// SIMATIC S7-200 project (STEP 7-Micro/WIN), CPU 224 UN REL 02.01

ORGANIZATION_BLOCK 主程序:OB1
TITLE=程序注释
BEGIN
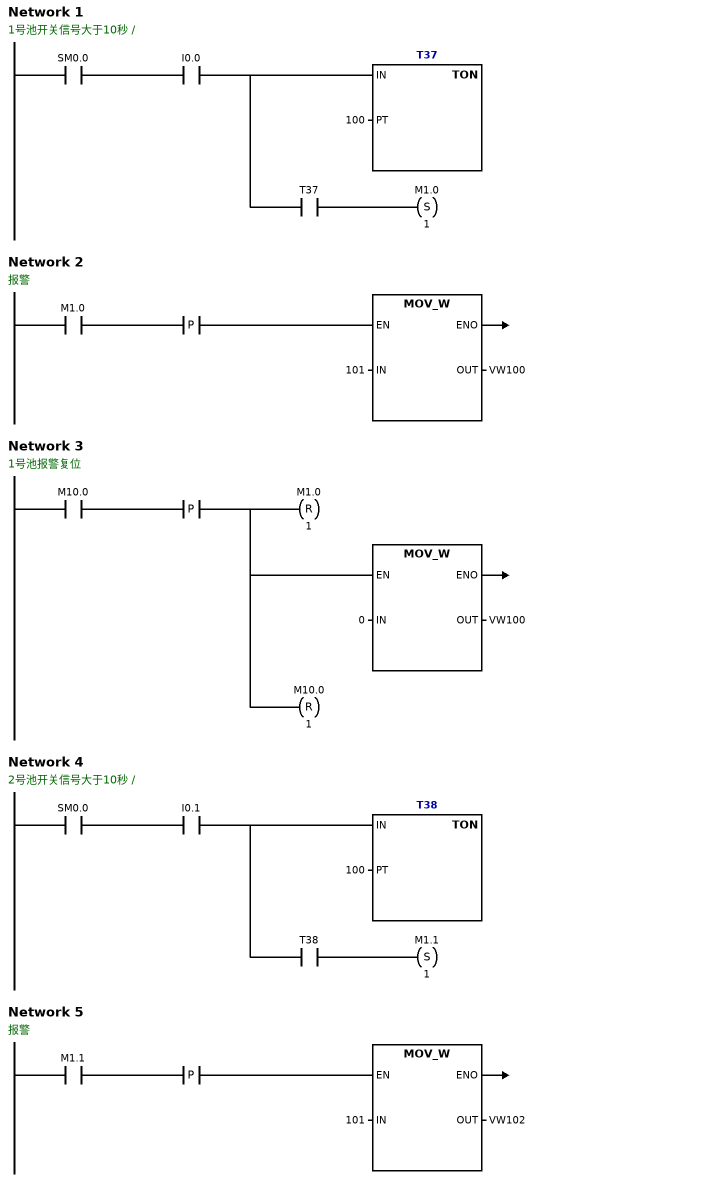
Network 1
// 1号池开关信号大于10秒
// 
LD     SM0.0
A      I0.0
TON    T37, 100
A      T37
S      M1.0, 1
Network 2 // 

// 报警
LD     M1.0
EU
MOVW   101, VW100
Network 3
// 1号池报警复位
LD     M10.0
EU
R      M1.0, 1
MOVW   0, VW100
R      M10.0, 1
Network 4
// 2号池开关信号大于10秒
// 
LD     SM0.0
A      I0.1
TON    T38, 100
A      T38
S      M1.1, 1
Network 5 // 

// 报警
LD     M1.1
EU
MOVW   101, VW102
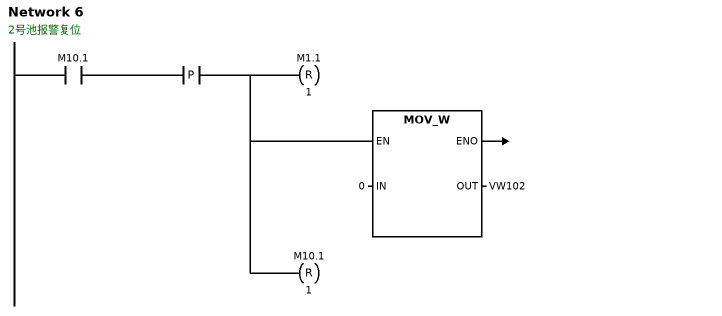
Network 6
// 2号池报警复位
LD     M10.1
EU
R      M1.1, 1
MOVW   0, VW102
R      M10.1, 1
END_ORGANIZATION_BLOCK

// SBR1: protected block, not included

// SBR2: protected block, not included

// SBR3: protected block, not included

// SBR4: protected block, not included
